// TIA Portal V20 export
// export: Created 2025-12-01T14:57:05.752345Z, ExportSetting None, DisplayName Totally Integrated Automation Portal, DisplayVersion V20 Update 3, DisplayName TIA Portal Openness, DisplayVersion V20 Update 3, DisplayName TIA Portal Version Control Interface, DisplayVersion V20 Update 3, DisplayName STEP 7 Professional, DisplayVersion V20 Update 3, DisplayName STEP 7 Safety, DisplayVersion V20 Update 2, DisplayName WinCC Basic/Comfort/Advanced, DisplayVersion V20 Update 3, DisplayName WinCC Professional, DisplayVersion V20 Update 3, DisplayName WinCC Unified, DisplayVersion V20 Update 3
FUNCTION "FC897_Generar_PointerAny" : Void   // FC897, LAD
{ S7_Optimized_Access := 'FALSE' }
AUTHOR : TRACKING
NAME : 20130301
VERSION : 3.0
// stored: AutoNumber false, SetENOAutomatically false
   VAR_INPUT
      TYP : Byte;   // 10h for S7
      DataTyp : Byte;   // 00=NullPoint,01=BOOL,02=BYTE,03=CHAR,04=WORD,05=INT,06=DWORD,07=DINT,08=REAL...
      repeatcounter : UDInt;   // amount of Bytes in Any Pointer
      DB_Number : UInt;   // Number of DB's
      storearea : Byte;   // 81=E-Input 82=A-Output 83=M-Flag 84=DB Datablock 85=DI-I-Datab.....
      storeaddresse : DWord;   // Byteaddress and Bitaddress
   END_VAR
   VAR_OUTPUT
      Any_Pointer : Any;   // result
   END_VAR
BEGIN

NETWORK
TITLE = 
      L     P##Any_Pointer;
      LAR1;

NETWORK
TITLE = Check Typ = S7 Value
      L     #TYP;
      L     B#16#10;  // This parameter has to be = 10h für S7
      <>I;
      BEC;
      T     B [AR1, P#0.0];  // write in Any-Pointer

NETWORK
TITLE = DatenTyp
      L     #DataTyp;
      JL    BEA1;  // in case of fault
      JU    WEIT;  // case is not possible
      JU    WEIT;  // TYPE BOOL       01
      JU    WEIT;  // TYPE BYTE       02
      JU    WEIT;  // TYPE CHAR       03
      JU    WEIT;  // TYPE WORD       04
      JU    WEIT;  // TYPE INT        05
      JU    WEIT;  // TYPE DWORD      06
      JU    WEIT;  // TYPE DINT       07
      JU    WEIT;  // TYPE REAL       08
      JU    WEIT;  // TYPE DATE       09
      JU    WEIT;  // TYPE TOD        0A
      JU    WEIT;  // TYPE TIME       0B
      JU    WEIT;  // TYPE S5TIME     0C
      JU    BEA1;  // RESERVED           0D
      JU    WEIT;  // TYPE DT         0E
      JU    BEA1;  // RESERVED           0F
      JU    BEA1;  // RESERVED           10
      JU    BEA1;  // RESERVED           11
      JU    BEA1;  // RESERVED           12
      JU    WEIT;  // TYPE STRING     13
      JU    BEA1;  // RESERVED           14
      JU    BEA1;  // RESERVED           15
      JU    BEA1;  // RESERVED           16
      JU    WEIT;  // TYPE BLOCK_FB   17
      JU    WEIT;  // TYPE BLOCK_FC   18
      JU    WEIT;  // TYPE BLOCK_DB   19
      JU    WEIT;  // TYPE BLOCK_SDB  1A
      JU    BEA1;  // RESERVED           1B
      JU    WEIT;  // TYPE COUNTER    1C
      JU    WEIT;  // TYPE TIMER      1D

BEA1: BEU;
WEIT: T     B [AR1, P#1.0];  // Datentyp

NETWORK
TITLE = write repeatcounter in Any Pointer
      L     #repeatcounter;
      T     W [AR1, P#2.0];

NETWORK
TITLE = write DB Number in Any Pointer
      L     #DB_Number;
      T     W [AR1, P#4.0];

NETWORK
TITLE = write storearea in Any Pointer
      L     #storeaddresse;
      L     DW#16#FFFFFF;  // Bereich ausmaskieren
      AD;
      T     D [AR1, P#6.0];  // BYTE 1

NETWORK
TITLE = write storaddresse in Any Pointer an match with storearea
      L     #storearea;
      L     B#16#F;  //hex: 8x mask out
      AW;
      JL    BEA2;

      JU    BEA2;  // zero not exist
      JU    NXT1;  // SP81: I input area
      JU    NXT1;  // SP82: Q output area
      JU    NXT1;  // SP83: M storearea flag
      JU    NXT1;  // SP84: DB Datenblock
      JU    NXT1;  // SP85: DI Instanz-Datenblock
      JU    NXT1;  // SP86: L-Stack 87=V previous Lokalstack
BEA2: BEU;  // Failur
NXT1: L     DW#16#80;
      OW;
      SLD   24;  // put storearea on right place in doubleword
      L     D [AR1, P#6.0];  // match pointer and area
      OD;
      T     D [AR1, P#6.0];  // -> result

NETWORK
TITLE = Watch in online mode to see the result
      L     B [AR1, P#0.0];
      L     B [AR1, P#1.0];
      L     W [AR1, P#2.0];
      L     W [AR1, P#4.0];
      L     D [AR1, P#6.0];
END_FUNCTION
